// TIA Portal V20 export
TYPE "UserDiag_typeSlot"
TITLE = UserDiag_typeSlot
   STRUCT
      hardwareId { ExternalAccessible := 'False'; ExternalVisible := 'False'; ExternalWritable := 'False'} : HW_IO := 16#0000;   // Hardware identifier of the module which is inserted in the slot
      state { ExternalAccessible := 'False'; ExternalVisible := 'False'; ExternalWritable := 'False'} : USInt := 0;   // Status of the device/slave. 1:ok; 2:faulty, 3:lost connection, 4:disabled, 5:problem, 12:was faulty, 13:was lost, 14:was disabled, 15:problem gone
      exists { ExternalAccessible := 'False'; ExternalVisible := 'False'; ExternalWritable := 'False'} : Bool := FALSE;   // TRUE: Modul is existing
      configured { ExternalAccessible := 'False'; ExternalVisible := 'False'; ExternalWritable := 'False'} : Bool := FALSE;   // TRUE: Modul is configured
      faulty { ExternalAccessible := 'False'; ExternalVisible := 'False'; ExternalWritable := 'False'} : Bool := FALSE;   // TRUE: Modul is faulty
      problem { ExternalAccessible := 'False'; ExternalVisible := 'False'; ExternalWritable := 'False'} : Bool := FALSE;   // TRUE: Modul has a problem
      disabled { ExternalAccessible := 'False'; ExternalVisible := 'False'; ExternalWritable := 'False'} : Bool := FALSE;   // TRUE: Modul is disabled
      error { ExternalAccessible := 'False'; ExternalVisible := 'False'; ExternalWritable := 'False'} : Bool := FALSE;   // TRUE: Error in module which is inserted in the slot
   END_STRUCT;
END_TYPE
